// TwinCAT 3 PLC project PLC
// ProgramVersion: 3.1.4024.0
// libraries:
//   EfficientIO Communicator, * (EfficientIO)
//   EfficientIO Energy Basic, * (EfficientIO)
//   EfficientIO ModbusTCP, * (EfficientIO)
//   Lynus Energy ModbusRTU, * (Lynus AG)
//   Lynus Persistent Data V1, * (Lynus AG)
//   Lynus Standards, * (EfficientIO)
//   Tc2_Math, * (Beckhoff Automation GmbH)
//   Tc2_MBus, * (Beckhoff Automation GmbH)
//   Tc2_Standard, * (Beckhoff Automation GmbH)
//   Tc2_System, * (Beckhoff Automation GmbH)
//   Tc2_Utilities, * (Beckhoff Automation GmbH)
//   Tc3_JsonXml, * (Beckhoff Automation GmbH)
//   Tc3_Module, * (Beckhoff Automation GmbH)
// project tree:
//   / Fast_Task.TcTTO, Middle_Task.TcTTO, Slow_Task.TcTTO (not stored)
//   FB/ FB_CoE_EL3443.TcPOU (not stored), FB_EM_Beckhoff_EL3443.TcPOU (not stored), FB_TimeSwitch_V2.TcPOU
//   POUs/ prgComEffIO.TcPOU, prgEM.TcPOU, prgEMS.TcPOU, prgGrid.TcPOU, prgHouse.TcPOU, prgPersistent.TcPOU (not stored), prgRWEffIO.TcPOU (not stored), prgSystemTime.TcPOU (not stored), prgVarEffIO.TcPOU (not stored)
// real-time tasks:
//   TASK Fast_Task: cycle T#8ms, priority 8, ADS port 350
//   TASK Middle_Task: cycle T#10ms, priority 10, ADS port 351
//   TASK Slow_Task: cycle T#20ms, priority 20, ADS port 352
// I/O:
//   DEVICE Gerät 1 (Beckhoff CCAT)
//   DEVICE Gerät 2 (EtherCAT), AmsNetId 5.100.32.125.3.1
//     Klemme 1 (EK1200) [EK1200-5000 EtherCAT Netzteil (2A E-Bus)]
//       Klemme 2 (EL3443) [EL3443 3K. Leistungsmessung]
//       Klemme 3 (EL2652) [EL2652 2K. Relais Ausgang, Wechsler (230V AC / 30V DC)]
//       Klemme 4 (EL2652) [EL2652 2K. Relais Ausgang, Wechsler (230V AC / 30V DC)]
//       Klemme 5 (EL2652) [EL2652 2K. Relais Ausgang, Wechsler (230V AC / 30V DC)]
//       Klemme 6 (EL2652) [EL2652 2K. Relais Ausgang, Wechsler (230V AC / 30V DC)]
//       Klemme 7 (EL9011) [EL9011 Endklemme]
// variable links:
//   PLC/PLC Instance <-> Device 2 (EtherCAT)/Term 1 (EK1200)/Term 2 (EL3443)
//     Middle_Task Inputs/prgGrid.lrActivePowerTotal <-> Total Active/Active Power
//     Middle_Task Inputs/prgGrid.lrGrid_Current_L1 <-> L1 Basic/Current
//     Middle_Task Inputs/prgGrid.lrGrid_Current_L2 <-> L2 Basic/Current
//     Middle_Task Inputs/prgGrid.lrGrid_Current_L3 <-> L3 Basic/Current
//     Middle_Task Inputs/prgGrid.lrGrid_Power_L1 <-> L1 Power/Active Power
//     Middle_Task Inputs/prgGrid.lrGrid_Power_L2 <-> L2 Power/Active Power
//     Middle_Task Inputs/prgGrid.lrGrid_Power_L3 <-> L3 Power/Active Power
//     Middle_Task Inputs/prgGrid.lrGrid_Voltage_L1 <-> L1 Basic/Voltage
//     Middle_Task Inputs/prgGrid.lrGrid_Voltage_L2 <-> L2 Basic/Voltage
//     Middle_Task Inputs/prgGrid.lrGrid_Voltage_L3 <-> L3 Basic/Voltage
//   PLC/PLC Instance <-> Device 2 (EtherCAT)/Term 1 (EK1200)/Term 3 (EL2652)
//     Middle_Task Outputs/prgEM.Boiler <-> Channel 2/Output
//     Middle_Task Outputs/prgEM.KaffeMaschine <-> Channel 1/Output
//   PLC/PLC Instance <-> Device 2 (EtherCAT)/Term 1 (EK1200)/Term 4 (EL2652)
//     Middle_Task Outputs/prgEM.Heizregister <-> Channel 2/Output
//     Middle_Task Outputs/prgEM.Reklame <-> Channel 1/Output
//   PLC/PLC Instance <-> Device 2 (EtherCAT)/Term 1 (EK1200)/Term 5 (EL2652)
//     Middle_Task Outputs/prgEM.Abluft <-> Channel 2/Output
//     Middle_Task Outputs/prgEM.Zuluft <-> Channel 1/Output

CONFIGURATION PLC
    RESOURCE PLC ON TwinCAT3
        TASK Fast_Task(INTERVAL := T#8ms, PRIORITY := 8);
        TASK Middle_Task(INTERVAL := T#10ms, PRIORITY := 10);
        PROGRAM prgVarEffIO WITH Fast_Task : prgVarEffIO;
        PROGRAM prgRWEffIO WITH Fast_Task : prgRWEffIO;
        PROGRAM prgPersistent WITH Middle_Task : prgPersistent;
        PROGRAM prgGrid WITH Middle_Task : prgGrid;
        PROGRAM prgEM WITH Middle_Task : prgEM;
    END_RESOURCE
END_CONFIGURATION

// ---- POUs/prgGrid.TcPOU
PROGRAM prgGrid
VAR
	fbKBusState					: FB_K_Bus_State;
	fbGrid						: FB_EM_Beckhoff_KL3403;
	uint_KBusState				: UINT;							//{#lynus.ag#()}
	fbGridCounter				: FB_EnergyCounter;
	lrGridPower					: LREAL;								//{#lynus.ag#()}
	lrVoltage_L1N				: LREAL;								//{#lynus.ag#()}
	lrVoltage_L2N				: LREAL;								//{#lynus.ag#()}
	lrVoltage_L3N				: LREAL;								//{#lynus.ag#()}
	
	lrGrid_Voltage_L1  	AT %I* 	: REAL;									//{#lynus.ag#()}
    lrGrid_Current_L1 	AT %I* 	: REAL;									//{#lynus.ag#()}
	lrGrid_Power_L1		AT %I* 	: REAL;									//{#lynus.ag#()}
	lrGrid_Voltage_L2  	AT %I* 	: REAL;									//{#lynus.ag#()}
    lrGrid_Current_L2 	AT %I* 	: REAL;									//{#lynus.ag#()}
	lrGrid_Power_L2		AT %I* 	: REAL;									//{#lynus.ag#()}
	lrGrid_Voltage_L3  	AT %I* 	: REAL;									//{#lynus.ag#()}
    lrGrid_Current_L3 	AT %I* 	: REAL;									//{#lynus.ag#()}
	lrGrid_Power_L3		AT %I* 	: REAL;									//{#lynus.ag#()}
	lrActivePowerTotal	AT %I*	: REAL;									//{#lynus.ag#()}
	

	Test : REAL;

	Grid_Voltage_L1  	: REAL;						

END_VAR
VAR PERSISTENT
	rSizeGridConn				: REAL;									//{#lynus.ag#()}
	lrCounterGridProd			: LREAL;								//{#lynus.ag#()}
	lrCounterGridCons			: LREAL;								//{#lynus.ag#()}
END_VAR

//The mapping of this function must be linked with the K-Bus State in the E/A Part
fbKBusState(	uiKBusState_OUT=> , 
				b_Kbus_notOk=> , 
				word_ErrorCount=> );
				
//Variablen werden verwendet -> Middle Task
Test:= lrGrid_Voltage_L1;
Test:= lrGrid_Current_L1;
Test:= lrGrid_Power_L1;
Test:= lrGrid_Voltage_L2;
Test:= lrGrid_Current_L2;
Test:= lrGrid_Power_L2;
Test:= lrGrid_Voltage_L3;
Test:= lrGrid_Current_L3;
Test:= lrGrid_Power_L3;
Test:= lrActivePowerTotal;

//The mapping of this function must be linked with the KL3443 in the E/A Part
//UV1
fbGrid(
	bEnable:= FALSE, 
	bChannel1Invers:= FALSE,				//Invert power data when transformer are mounted upside down
	bChannel2Invers:= FALSE,				// CT seems to be wired the wrong wy around
	bChannel3Invers:= FALSE,
	uiCurrentTransformerRatioL1:= 300, 		//Transformer ratio on the secondary side
	uiCurrentTransformerRatioL2:= 300, 
	uiCurrentTransformerRatioL3:= 300, 
	uiKBusState_IN:= fbKBusState.uiKBusState_OUT, 
	stDataEMPower=> , 
	stDataEMCounter=> , 
	stDataEMPowerRealTime=> , 
	stDataEMCounterRealTime=> , 
	diNrOfEM_OUT=> );
	
uint_KBusState 	:=	fbKBusState.uiKBusState_OUT;
lrGridPower 	:= 	lrActivePowerTotal/1000;

// EnergyCounter
fbGridCounter(
	byActiveTariff:= 1, 
	lrPowerInput:= lrGridPower, 
	lrTotalCounterEnergy_Consumption=> , 
	lrTotalCounterEnergy_Production=> , 
	lrCounterEnergyT1_Consumption=> , 
	lrCounterEnergyT2_Consumption=> , 
	lrCounterEnergyT1_Production=> , 
	lrCounterEnergyT2_Production=> );

IF fbGridCounter.lrTotalCounterEnergy_Production > lrCounterGridProd THEN  	
		lrCounterGridProd := fbGridCounter.lrTotalCounterEnergy_Production;
END_IF

IF fbGridCounter.lrTotalCounterEnergy_Consumption > lrCounterGridCons THEN  	
	lrCounterGridCons := fbGridCounter.lrTotalCounterEnergy_Consumption;
END_IF

lrVoltage_L1N := fbGrid.stDataEMPower.lrVoltageL1N;
lrVoltage_L2N := fbGrid.stDataEMPower.lrVoltageL2N;
lrVoltage_L3N := fbGrid.stDataEMPower.lrVoltageL3N;

END_PROGRAM

// ---- POUs/prgEM.TcPOU
PROGRAM prgEM
VAR
	//Eingangsvariable: Aktueller Leistungswert aus prgGrid
    PowerValue 				: REAL := prgGrid.lrGridPower;
	Threshold 				: REAL := 35.0;  				//Schwelle zum Abschalten
	//Hysterese zum Vermeiden von schnellen Ein-/Ausschaltvorgängen
    Hysteresis 				: REAL := 5.0;
	//Zustandsvariablen zur Vermeidung von Schwingungen
    BoilerActive	 		: BOOL := TRUE;
    ReklameActive	 		: BOOL := TRUE;
	HeizregisterActive		: BOOL := TRUE;
    ZuluftActive	 		: BOOL := TRUE;
	AbluftActive	 		: BOOL := TRUE;
	//RELAI 1
	KaffeMaschine  	AT %Q* 	: BOOL;
	Boiler  		AT %Q* 	: BOOL;
	//RELAI 2
	Reklame  		AT %Q* 	: BOOL;
	Heizregister	AT %Q* 	: BOOL;
	//RELAI 3
	Zuluft  		AT %Q* 	: BOOL;
	Abluft	 		AT %Q* 	: BOOL;
	//RELAI 4 - OFFEN (Keine Anschlüsse)
	//RELAI4_CH1		AT %Q* 	: BOOL;
	//RELAI4_CH2		AT %Q* 	: BOOL;
	
	Test					:BOOL;
	
END_VAR

Test := KaffeMaschine;
Test := Boiler;
Test := Reklame;
Test := Heizregister;
Test := Zuluft;
Test := Abluft;
(* Logik zum Lastenmanagement mit einem Schwellenwert *)

(* Relais 1 CH 2 - Einschalten *)
IF PowerValue > Threshold AND BoilerActive THEN
    Boiler 			:= TRUE; 							//Relai wird eingeschalten um die Verbindung zu öffnen
    BoilerActive 	:= FALSE;
ELSIF PowerValue < (Threshold - Hysteresis) AND NOT BoilerActive THEN
    Boiler 			:= FALSE;  
    BoilerActive 	:= TRUE;
END_IF;
(*
(* Relais 2 CH1 - Einschalten *)
IF PowerValue > Threshold AND ReklameActive THEN
    Reklame 		:= TRUE; (* Relais 2 einschalten *)
    ReklameActive 	:= FALSE;
ELSIF PowerValue < (Threshold - Hysteresis) AND NOT ReklameActive THEN
    Reklame			:= FALSE;  (* Relais 2 ausschalten *)
    ReklameActive 	:= TRUE;
END_IF;
*)
(* Relais 2 CH2 - Einschalten *)
IF PowerValue > Threshold AND HeizregisterActive THEN
    Heizregister 		:= TRUE; (* Relais 2 einschalten *)
    HeizregisterActive 	:= FALSE;
ELSIF PowerValue < (Threshold - Hysteresis) AND NOT HeizregisterActive THEN
    Heizregister		:= FALSE;  (* Relais 2 ausschalten *)
    HeizregisterActive 	:= TRUE;
END_IF;

(* Relais 3 CH1 & CH2 - Einschalten *)
IF PowerValue > Threshold AND ZuluftActive AND AbluftActive THEN
    Zuluft := TRUE;
	Abluft := TRUE;
    ZuluftActive := FALSE;
	AbluftActive := FALSE;
ELSIF PowerValue < (Threshold - Hysteresis) AND NOT ZuluftActive AND NOT AbluftActive THEN
    Zuluft := FALSE;
	Abluft := FALSE;
	ZuluftActive := TRUE;
	AbluftActive := TRUE;
END_IF;

END_PROGRAM

// ---- FB/FB_TimeSwitch_V2.TcPOU
FUNCTION_BLOCK FB_TimeSwitch_V2
VAR_INPUT
	b_Enable: BOOL;
	b_StatusOn: BOOL;
	structSystemTime: timestruct;
	byte_MoFr_Open_Hour: BYTE;
	byte_MoFr_Open_Minute: BYTE;
	byte_MoFr_Close_Hour: BYTE;
	byte_MoFr_Close_Minute: BYTE;
	byte_Sa_Open_Hour: BYTE;
	byte_Sa_Open_Minute: BYTE;
	byte_Sa_Close_Hour: BYTE;
	byte_Sa_Close_Minute: BYTE;	
	byte_So_Open_Hour: BYTE;
	byte_So_Open_Minute: BYTE;
	byte_So_Close_Hour: BYTE;
	byte_So_Close_Minute: BYTE;
	real_Offset_Start: REAL;
	real_Offset_Stop: REAL;	
	b_On_Manual: BOOL;
	b_Off_Manual: BOOL;
END_VAR
VAR_OUTPUT
	b_Output_On: BOOL;
	b_Error: BOOL;
END_VAR
VAR
	TON_0: ton;
	byte_Day :BYTE;		// 0: Sunday, 1: Monday,....
	time_now             		: TIME;
	time_MoFr_Open             	: TIME;
	time_MoFr_Close             : TIME;
	time_Sa_Open             	: TIME;
	time_Sa_Close             	: TIME;
	time_So_Open             	: TIME;
	time_So_Close             	: TIME;
	

	RS_0: rs;
	R_TRIG_0: r_trig;
	R_TRIG_1: r_trig;
	dt_Test: DATE_AND_TIME;
	tod_test: TIME_OF_DAY;
	time_temp: TIME;
	time_Start_MoFr_Calc: TIME;
	time_Stop_MoFr_Calc: TIME;
	time_Start_Sa_Calc: TIME;
	time_Stop_Sa_Calc: TIME;
	time_Start_So_Calc: TIME;
	time_Stop_So_Calc: TIME;
	
	FB_WeeklyTimeSwitch_MoFr: FB_WeeklyTimeSwitch;
	FB_WeeklyTimeSwitch_Sa: FB_WeeklyTimeSwitch;
	FB_WeeklyTimeSwitch_So: FB_WeeklyTimeSwitch;
	RS_manu: rs;
	b_Auto_on: BOOL;

	R_TRIG_2: r_trig;
	R_TRIG_3: r_trig;
	F_TRIG_0: f_trig;
	R_TRIG_4: r_trig;
	R_TRIG_FirstCycle: r_trig;
	time_Zero             	: TIME;
	
END_VAR
VAR // added by the converter: edge detectors and wires of the graphical bodies
    _w1 : DATE_AND_TIME;
    _w2 : TIME_OF_DAY;
    _w3 : BOOL;
END_VAR

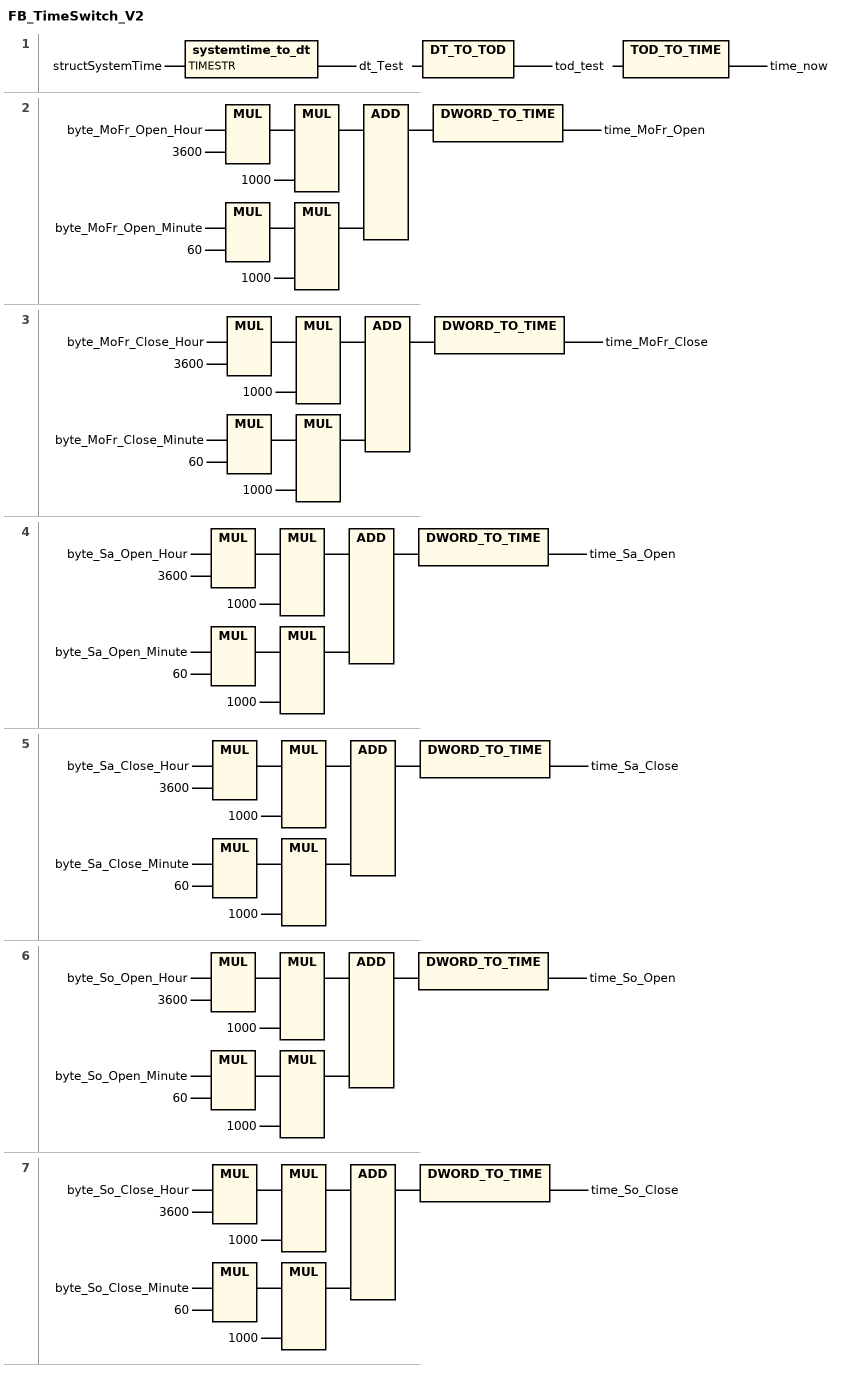
// NETWORK 1
_w1 := systemtime_to_dt(TIMESTR := structSystemTime);
dt_Test := _w1;
_w2 := DT_TO_TOD(_w1);
tod_test := _w2;
time_now := TOD_TO_TIME(_w2);

// NETWORK 2
time_MoFr_Open := DWORD_TO_TIME((byte_MoFr_Open_Hour * 3600) * 1000 + (byte_MoFr_Open_Minute * 60) * 1000);

// NETWORK 3
time_MoFr_Close := DWORD_TO_TIME((byte_MoFr_Close_Hour * 3600) * 1000 + (byte_MoFr_Close_Minute * 60) * 1000);

// NETWORK 4
time_Sa_Open := DWORD_TO_TIME((byte_Sa_Open_Hour * 3600) * 1000 + (byte_Sa_Open_Minute * 60) * 1000);

// NETWORK 5
time_Sa_Close := DWORD_TO_TIME((byte_Sa_Close_Hour * 3600) * 1000 + (byte_Sa_Close_Minute * 60) * 1000);

// NETWORK 6
time_So_Open := DWORD_TO_TIME((byte_So_Open_Hour * 3600) * 1000 + (byte_So_Open_Minute * 60) * 1000);

// NETWORK 7
time_So_Close := DWORD_TO_TIME((byte_So_Close_Hour * 3600) * 1000 + (byte_So_Close_Minute * 60) * 1000);

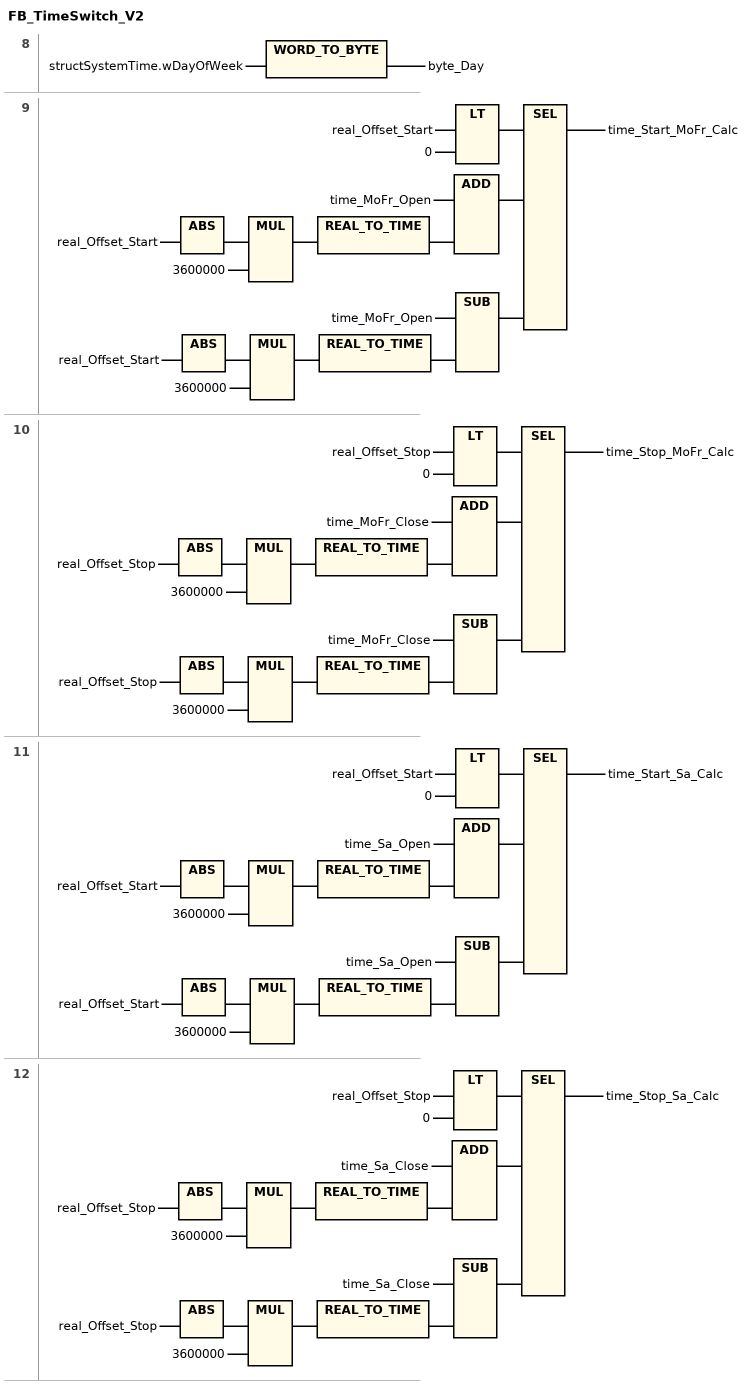
// NETWORK 8
byte_Day := WORD_TO_BYTE(structSystemTime.wDayOfWeek);

// NETWORK 9
time_Start_MoFr_Calc := SEL(real_Offset_Start < 0, time_MoFr_Open + REAL_TO_TIME(ABS(real_Offset_Start) * 3600000), time_MoFr_Open - REAL_TO_TIME(ABS(real_Offset_Start) * 3600000));

// NETWORK 10
time_Stop_MoFr_Calc := SEL(real_Offset_Stop < 0, time_MoFr_Close + REAL_TO_TIME(ABS(real_Offset_Stop) * 3600000), time_MoFr_Close - REAL_TO_TIME(ABS(real_Offset_Stop) * 3600000));

// NETWORK 11
time_Start_Sa_Calc := SEL(real_Offset_Start < 0, time_Sa_Open + REAL_TO_TIME(ABS(real_Offset_Start) * 3600000), time_Sa_Open - REAL_TO_TIME(ABS(real_Offset_Start) * 3600000));

// NETWORK 12
time_Stop_Sa_Calc := SEL(real_Offset_Stop < 0, time_Sa_Close + REAL_TO_TIME(ABS(real_Offset_Stop) * 3600000), time_Sa_Close - REAL_TO_TIME(ABS(real_Offset_Stop) * 3600000));

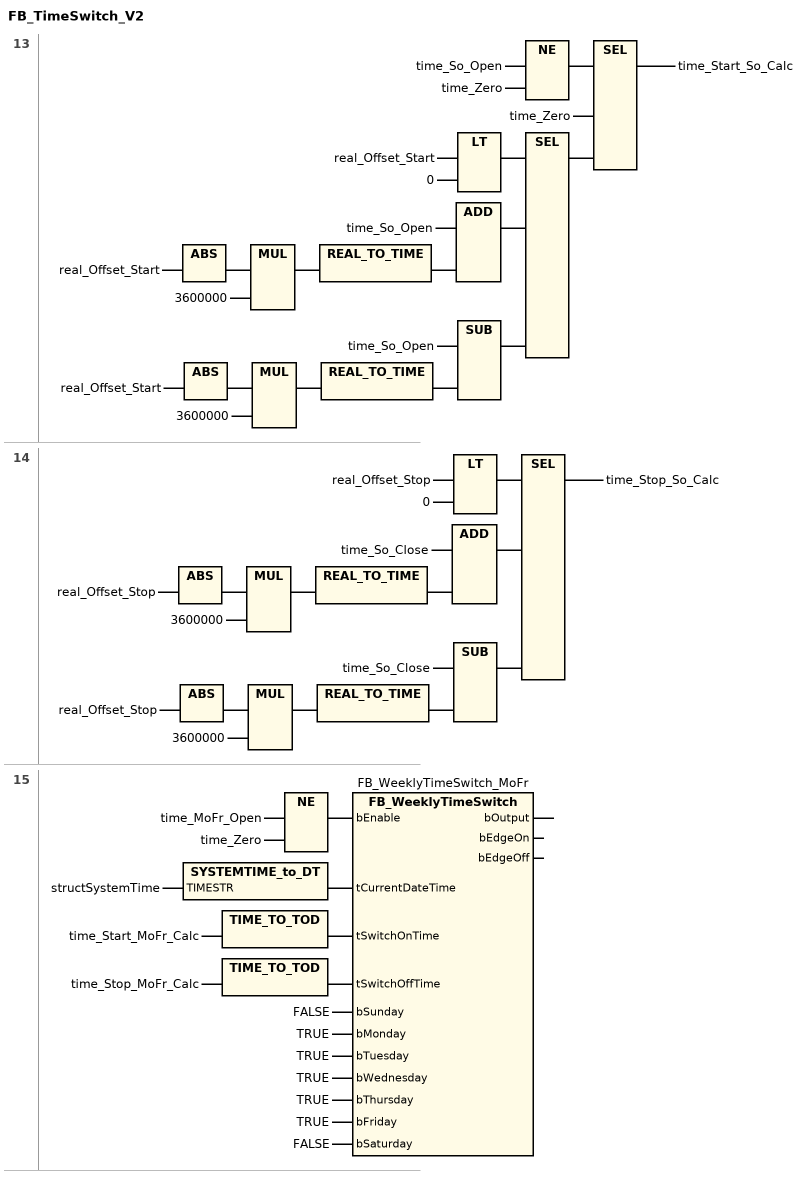
// NETWORK 13
time_Start_So_Calc := SEL(time_So_Open <> time_Zero, time_Zero, SEL(real_Offset_Start < 0, time_So_Open + REAL_TO_TIME(ABS(real_Offset_Start) * 3600000), time_So_Open - REAL_TO_TIME(ABS(real_Offset_Start) * 3600000)));

// NETWORK 14
time_Stop_So_Calc := SEL(real_Offset_Stop < 0, time_So_Close + REAL_TO_TIME(ABS(real_Offset_Stop) * 3600000), time_So_Close - REAL_TO_TIME(ABS(real_Offset_Stop) * 3600000));

// NETWORK 15
FB_WeeklyTimeSwitch_MoFr(
    bEnable := time_MoFr_Open <> time_Zero,
    tCurrentDateTime := SYSTEMTIME_to_DT(TIMESTR := structSystemTime),
    tSwitchOnTime := TIME_TO_TOD(time_Start_MoFr_Calc),
    tSwitchOffTime := TIME_TO_TOD(time_Stop_MoFr_Calc),
    bSunday := FALSE,
    bMonday := TRUE,
    bTuesday := TRUE,
    bWednesday := TRUE,
    bThursday := TRUE,
    bFriday := TRUE,
    bSaturday := FALSE); // FB_WeeklyTimeSwitch

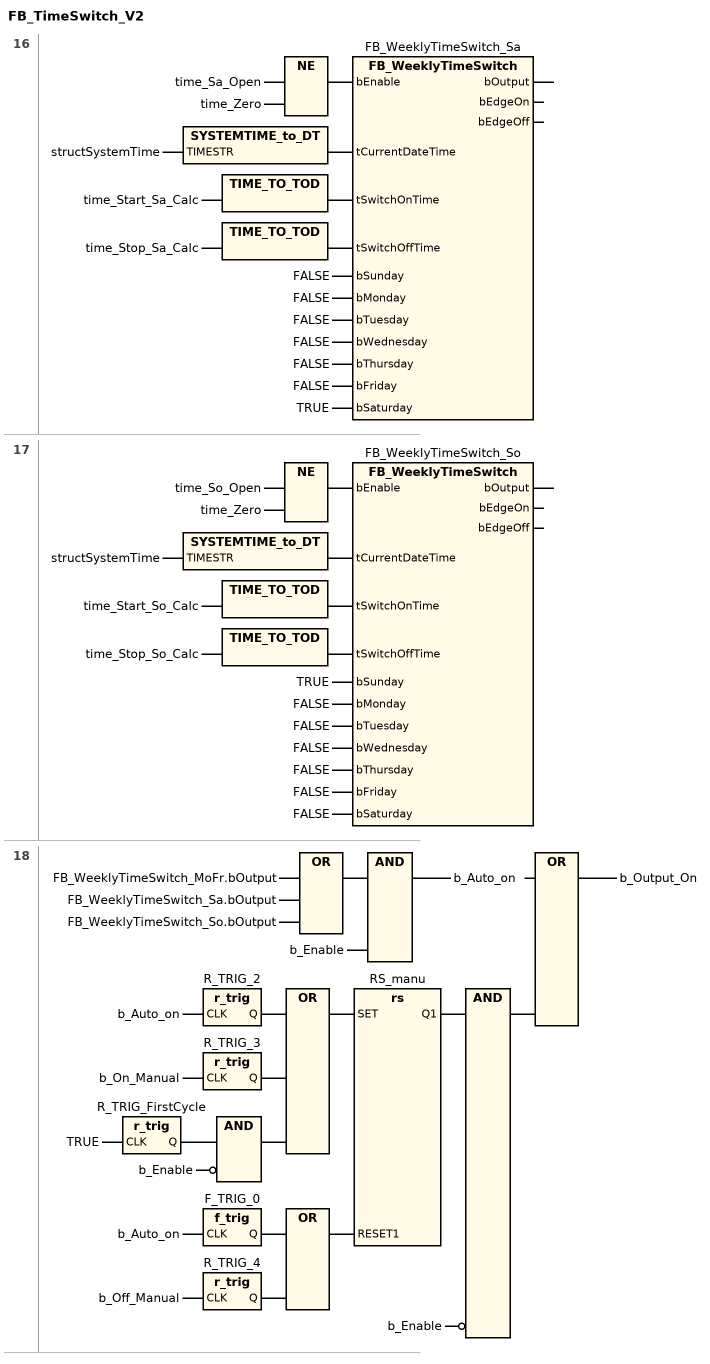
// NETWORK 16
FB_WeeklyTimeSwitch_Sa(
    bEnable := time_Sa_Open <> time_Zero,
    tCurrentDateTime := SYSTEMTIME_to_DT(TIMESTR := structSystemTime),
    tSwitchOnTime := TIME_TO_TOD(time_Start_Sa_Calc),
    tSwitchOffTime := TIME_TO_TOD(time_Stop_Sa_Calc),
    bSunday := FALSE,
    bMonday := FALSE,
    bTuesday := FALSE,
    bWednesday := FALSE,
    bThursday := FALSE,
    bFriday := FALSE,
    bSaturday := TRUE); // FB_WeeklyTimeSwitch

// NETWORK 17
FB_WeeklyTimeSwitch_So(
    bEnable := time_So_Open <> time_Zero,
    tCurrentDateTime := SYSTEMTIME_to_DT(TIMESTR := structSystemTime),
    tSwitchOnTime := TIME_TO_TOD(time_Start_So_Calc),
    tSwitchOffTime := TIME_TO_TOD(time_Stop_So_Calc),
    bSunday := TRUE,
    bMonday := FALSE,
    bTuesday := FALSE,
    bWednesday := FALSE,
    bThursday := FALSE,
    bFriday := FALSE,
    bSaturday := FALSE); // FB_WeeklyTimeSwitch

// NETWORK 18
_w3 := (FB_WeeklyTimeSwitch_MoFr.bOutput OR FB_WeeklyTimeSwitch_Sa.bOutput OR FB_WeeklyTimeSwitch_So.bOutput) AND b_Enable;
b_Auto_on := _w3;
R_TRIG_2(CLK := b_Auto_on); // r_trig
R_TRIG_3(CLK := b_On_Manual); // r_trig
R_TRIG_FirstCycle(CLK := TRUE); // r_trig
F_TRIG_0(CLK := b_Auto_on); // f_trig
R_TRIG_4(CLK := b_Off_Manual); // r_trig
RS_manu(SET := R_TRIG_2.Q OR R_TRIG_3.Q OR R_TRIG_FirstCycle.Q AND NOT b_Enable, RESET1 := F_TRIG_0.Q OR R_TRIG_4.Q); // rs
b_Output_On := _w3 OR RS_manu.Q1 AND NOT b_Enable;

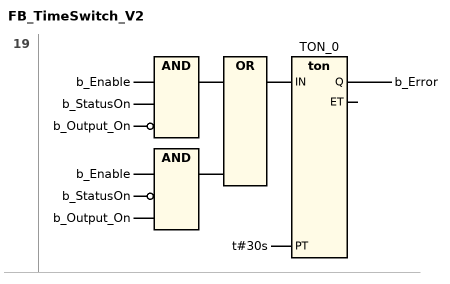
// NETWORK 19
TON_0(IN := b_Enable AND b_StatusOn AND NOT b_Output_On OR b_Enable AND NOT b_StatusOn AND b_Output_On, PT := t#30s); // ton
b_Error := TON_0.Q;

END_FUNCTION_BLOCK

// ---- POUs/prgComEffIO.TcPOU
PROGRAM prgComEffIO
VAR
	fbCom		: FB_MqttCommunicator_V5;
END_VAR

// CX-7BDACD
fbCom(
	bConnect:= TRUE, 
	strAuthKey := 'ENE87365342998',
	sUserName:= 'a4398363-713f-45e4-8f12-13b95d7f2606', 
	sUserPassword:= '196c948c-aabd-4764-8be4-f15873a2b8fa', 
	eSavePositionCertificate:= eSavePositionOnPLC.ePostionHardDisk,
	time_HeartBeat_sec:= T#50S, 
	bConnected=> , 
	bError=> , 
	hrErrorCode=> , 
	eConnectionState=> , 
	eErrorMessage_Out=> );

END_PROGRAM

// ---- POUs/prgEMS.TcPOU
PROGRAM prgEMS
VAR
	FB_TimeSwitch_CH1: FB_TimeSwitch_v2;
	FB_TimeSwitch_CH2: FB_TimeSwitch_v2;
	FB_TimeSwitch_CH3: FB_TimeSwitch_v2;
	FB_TimeSwitch_CH4: FB_TimeSwitch_v2;
	FB_TimeSwitch_CH5: FB_TimeSwitch_v2;	// outside light
	FB_TimeSwitch_CH6: FB_TimeSwitch_v2;	// Coffee maschine
	FB_TimeSwitch_CH7: FB_TimeSwitch_v2;	// Ventilation
	FB_TimeSwitch_CH8: FB_TimeSwitch_v2;	// Coffee maschine2
	
	b_Manual_On_CH1		: BOOL;						//{#lynus.ag#()}
	b_Manual_Off_CH1	: BOOL;						//{#lynus.ag#()}
	b_Manual_On_CH2		: BOOL;						//{#lynus.ag#()}
	b_Manual_Off_CH2	: BOOL;						//{#lynus.ag#()}
	b_Manual_On_CH3		: BOOL;						//{#lynus.ag#()}
	b_Manual_Off_CH3	: BOOL;						//{#lynus.ag#()}
	b_Manual_On_CH4		: BOOL;						//{#lynus.ag#()}
	b_Manual_Off_CH4	: BOOL;						//{#lynus.ag#()}
	b_Manual_On_CH5		: BOOL;						//{#lynus.ag#()}
	b_Manual_Off_CH5	: BOOL;						//{#lynus.ag#()}
	b_Manual_On_Coffee_CH6		: BOOL;						//{#lynus.ag#()}
	b_Manual_Off_Coffee_CH6		: BOOL;						//{#lynus.ag#()}
	b_Manual_On_Vent_CH7		: BOOL;						//{#lynus.ag#()}
	b_Manual_Off_Vent_CH7		: BOOL;						//{#lynus.ag#()}
	b_Manual_On_Coffee2_CH8		: BOOL;						//{#lynus.ag#()}
	b_Manual_Off_Coffee2_CH8	: BOOL;						//{#lynus.ag#()}

	fbCalcSunriseSunset   		: FB_CalcSunriseSunset;
	todSunrise            		: TOD;
	todSunset             		: TOD;
	fb_GetTimeZoneInfo	:FB_GetTimeZoneInformation;
	b_firstCycle: BOOL;
	RS_Outsidelight: RS;
	r_trig_on: R_trig;
	r_trig_off: R_trig;
	b_Out_CH1: BOOL;
	b_Out_CH2: BOOL;
	b_Out_CH3: BOOL;
	b_Out_CH4: BOOL;
	b_Out_CH5: BOOL;
	b_Out_CH6: BOOL;
	b_Out_CH7: BOOL;		
	b_Out_CH8: BOOL;		
	b_LoadOn_CH1	: BOOL;						//{#lynus.ag#()}
	b_LoadOn_CH2	: BOOL;						//{#lynus.ag#()}
	b_LoadOn_CH3	: BOOL;						//{#lynus.ag#()}
	b_LoadOn_CH4	: BOOL;						//{#lynus.ag#()}
	b_LoadOn_CH5	: BOOL;						//{#lynus.ag#()}
	b_LoadOn_CH6	: BOOL;						//{#lynus.ag#()}
	b_LoadOn_CH7	: BOOL;						//{#lynus.ag#()}
	b_LoadOn_CH8	: BOOL;						//{#lynus.ag#()}
END_VAR
VAR_INPUT
	fDegreeOfLongitude 	:LREAL;
	fDegreeOfLatitude	:LREAL;
	b_Input_KeySwitch		: BOOL;						//{#lynus.ag#()}
	b_Input_Spare			: BOOL;						//{#lynus.ag#()}
	m_UnderGroundMode		: BOOL;						//{#lynus.ag#()}
	int_test:INT;
END_VAR
VAR PERSISTENT
// opening hours
	byte_MoFr_Open_Hour		:BYTE;					//{#lynus.ag#()}
	byte_MoFr_Open_Minute	:BYTE;					//{#lynus.ag#()}
	byte_MoFr_Close_Hour	:BYTE;					//{#lynus.ag#()}
	byte_MoFr_Close_Minute	:BYTE;					//{#lynus.ag#()}
	byte_Sa_Open_Hour		:BYTE;					//{#lynus.ag#()}
	byte_Sa_Open_Minute		:BYTE;					//{#lynus.ag#()}
	byte_Sa_Close_Hour		:BYTE;					//{#lynus.ag#()}
	byte_Sa_Close_Minute	:BYTE;					//{#lynus.ag#()}
	byte_So_Open_Hour		:BYTE;					//{#lynus.ag#()}
	byte_So_Open_Minute		:BYTE;					//{#lynus.ag#()}
	byte_So_Close_Hour		:BYTE;					//{#lynus.ag#()}
	byte_So_Close_Minute	:BYTE;					//{#lynus.ag#()}
// offset CH1 in hours			
	b_Enable_Control_CH1		:BOOL;				//{#lynus.ag#()}
	real_Offset_Start_CH1		:REAL;				//{#lynus.ag#()}
	real_Offset_Stop_CH1		:REAL;				//{#lynus.ag#()}
// offset CH2 in hours			
	b_Enable_Control_CH2		:BOOL;				//{#lynus.ag#()}
	real_Offset_Start_CH2		:REAL;				//{#lynus.ag#()}
	real_Offset_Stop_CH2		:REAL;				//{#lynus.ag#()}
// offset CH3 in hours			
	b_Enable_Control_CH3		:BOOL;				//{#lynus.ag#()}
	real_Offset_Start_CH3		:REAL;				//{#lynus.ag#()}
	real_Offset_Stop_CH3		:REAL;				//{#lynus.ag#()}
// offset CH4 in hours			
	b_Enable_Control_CH4		:BOOL;				//{#lynus.ag#()}
	real_Offset_Start_CH4		:REAL;				//{#lynus.ag#()}
	real_Offset_Stop_CH4		:REAL;				//{#lynus.ag#()}
// offset CH5 in hours			
	b_Enable_Control_CH5		:BOOL;				//{#lynus.ag#()}
	real_Offset_Start_CH5		:REAL;				//{#lynus.ag#()}
	real_Offset_Stop_CH5		:REAL;				//{#lynus.ag#()}
// offset CH6 in hours			
	b_Enable_Control_Coffee_CH6	:BOOL;				//{#lynus.ag#()}
	real_Offset_Start_Coffee_CH6:REAL;				//{#lynus.ag#()}
	real_Offset_Stop_Coffee_CH6	:REAL;				//{#lynus.ag#()}
// offset CH7 in hours			
	b_Enable_Control_Vent_CH7	:BOOL;				//{#lynus.ag#()}
	real_Offset_Start_CH7		:REAL;				//{#lynus.ag#()}
	real_Offset_Stop_CH7		:REAL;				//{#lynus.ag#()}
// offset CH8 in hours			
	b_Enable_Control_Coffee2_CH8	:BOOL;				//{#lynus.ag#()}
	real_Offset_Start_Coffee2_CH8	:REAL;				//{#lynus.ag#()}
	real_Offset_Stop_Coffee2_CH8	:REAL;				//{#lynus.ag#()}
END_VAR


FB_TimeSwitch_CH1(
	b_Enable:= b_Enable_Control_CH1, 
	b_StatusOn:= NOT b_Out_CH1, 
	structSystemTime:=prgSystemTime.structSystemTime , 
	byte_MoFr_Open_Hour:= byte_MoFr_Open_Hour , 
	byte_MoFr_Open_Minute:= byte_MoFr_Open_Minute, 
	byte_MoFr_Close_Hour:= byte_MoFr_Close_Hour , 
	byte_MoFr_Close_Minute:= byte_MoFr_Close_Minute, 
	byte_Sa_Open_Hour:= byte_Sa_Open_Hour, 
	byte_Sa_Open_Minute:= byte_Sa_Open_Minute , 
	byte_Sa_Close_Hour:= byte_Sa_Close_Hour , 
	byte_Sa_Close_Minute:= byte_Sa_Close_Minute, 
	byte_So_Open_Hour:= byte_So_Open_Hour, 
	byte_So_Open_Minute:= byte_So_Open_Minute, 
	byte_So_Close_Hour:= byte_So_Close_Hour, 
	byte_So_Close_Minute:= byte_So_Close_Minute, 
	real_Offset_Start:= real_Offset_Start_CH1 , 
	real_Offset_Stop:= real_Offset_Stop_CH1 , 
	b_On_Manual:= b_Manual_On_CH1, 
	b_Off_Manual:= b_Manual_Off_CH1, 
	b_Output_On=> b_LoadOn_CH1, 
	b_Error=> );
b_Out_CH1 := NOT FB_TimeSwitch_CH1.b_Output_On;

FB_TimeSwitch_CH2(
	b_Enable:= b_Enable_Control_CH2, 
	b_StatusOn:= NOT b_Out_CH2, 
	structSystemTime:=prgSystemTime.structSystemTime , 
	byte_MoFr_Open_Hour:= byte_MoFr_Open_Hour , 
	byte_MoFr_Open_Minute:= byte_MoFr_Open_Minute, 
	byte_MoFr_Close_Hour:= byte_MoFr_Close_Hour , 
	byte_MoFr_Close_Minute:= byte_MoFr_Close_Minute, 
	byte_Sa_Open_Hour:= byte_Sa_Open_Hour, 
	byte_Sa_Open_Minute:= byte_Sa_Open_Minute , 
	byte_Sa_Close_Hour:= byte_Sa_Close_Hour , 
	byte_Sa_Close_Minute:= byte_Sa_Close_Minute, 
	byte_So_Open_Hour:= byte_So_Open_Hour, 
	byte_So_Open_Minute:= byte_So_Open_Minute, 
	byte_So_Close_Hour:= byte_So_Close_Hour, 
	byte_So_Close_Minute:= byte_So_Close_Minute, 
	real_Offset_Start:= real_Offset_Start_CH2 , 
	real_Offset_Stop:= real_Offset_Stop_CH2 , 
	b_On_Manual:= b_Manual_On_CH2, 
	b_Off_Manual:= b_Manual_Off_CH2, 
	b_Output_On=> b_LoadOn_CH2, 
	b_Error=> );
b_Out_CH2 := NOT FB_TimeSwitch_CH2.b_Output_On;

FB_TimeSwitch_CH3(
	b_Enable:= b_Enable_Control_CH3, 
	b_StatusOn:= NOT b_Out_CH3, 
	structSystemTime:=prgSystemTime.structSystemTime , 
	byte_MoFr_Open_Hour:= byte_MoFr_Open_Hour , 
	byte_MoFr_Open_Minute:= byte_MoFr_Open_Minute, 
	byte_MoFr_Close_Hour:= byte_MoFr_Close_Hour , 
	byte_MoFr_Close_Minute:= byte_MoFr_Close_Minute, 
	byte_Sa_Open_Hour:= byte_Sa_Open_Hour, 
	byte_Sa_Open_Minute:= byte_Sa_Open_Minute , 
	byte_Sa_Close_Hour:= byte_Sa_Close_Hour , 
	byte_Sa_Close_Minute:= byte_Sa_Close_Minute, 
	byte_So_Open_Hour:= byte_So_Open_Hour, 
	byte_So_Open_Minute:= byte_So_Open_Minute, 
	byte_So_Close_Hour:= byte_So_Close_Hour, 
	byte_So_Close_Minute:= byte_So_Close_Minute, 
	real_Offset_Start:= real_Offset_Start_CH3 , 
	real_Offset_Stop:= real_Offset_Stop_CH3 , 
	b_On_Manual:= b_Manual_On_CH3, 
	b_Off_Manual:= b_Manual_Off_CH3, 
	b_Output_On=> b_LoadOn_CH3, 
	b_Error=> );
b_Out_CH3 := NOT FB_TimeSwitch_CH3.b_Output_On;
	
FB_TimeSwitch_CH4(
	b_Enable:= b_Enable_Control_CH4, 
	b_StatusOn:= NOT b_Out_CH4, 
	structSystemTime:=prgSystemTime.structSystemTime , 
	byte_MoFr_Open_Hour:= byte_MoFr_Open_Hour , 
	byte_MoFr_Open_Minute:= byte_MoFr_Open_Minute, 
	byte_MoFr_Close_Hour:= byte_MoFr_Close_Hour , 
	byte_MoFr_Close_Minute:= byte_MoFr_Close_Minute, 
	byte_Sa_Open_Hour:= byte_Sa_Open_Hour, 
	byte_Sa_Open_Minute:= byte_Sa_Open_Minute , 
	byte_Sa_Close_Hour:= byte_Sa_Close_Hour , 
	byte_Sa_Close_Minute:= byte_Sa_Close_Minute, 
	byte_So_Open_Hour:= byte_So_Open_Hour, 
	byte_So_Open_Minute:= byte_So_Open_Minute, 
	byte_So_Close_Hour:= byte_So_Close_Hour, 
	byte_So_Close_Minute:= byte_So_Close_Minute, 
	real_Offset_Start:= real_Offset_Start_CH4 , 
	real_Offset_Stop:= real_Offset_Stop_CH4 , 
	b_On_Manual:= b_Manual_On_CH4, 
	b_Off_Manual:= b_Manual_Off_CH4, 
	b_Output_On=> b_LoadOn_CH4 ,
	b_Error=> );
b_Out_CH4 := NOT FB_TimeSwitch_CH4.b_Output_On;
	
FB_TimeSwitch_CH5(
	b_Enable:= b_Enable_Control_CH5, 
	b_StatusOn:= NOT b_Out_CH5, 
	structSystemTime:=prgSystemTime.structSystemTime , 
	byte_MoFr_Open_Hour:= byte_MoFr_Open_Hour , 
	byte_MoFr_Open_Minute:= byte_MoFr_Open_Minute, 
	byte_MoFr_Close_Hour:= byte_MoFr_Close_Hour , 
	byte_MoFr_Close_Minute:= byte_MoFr_Close_Minute, 
	byte_Sa_Open_Hour:= byte_Sa_Open_Hour, 
	byte_Sa_Open_Minute:= byte_Sa_Open_Minute , 
	byte_Sa_Close_Hour:= byte_Sa_Close_Hour , 
	byte_Sa_Close_Minute:= byte_Sa_Close_Minute, 
	byte_So_Open_Hour:= byte_So_Open_Hour, 
	byte_So_Open_Minute:= byte_So_Open_Minute, 
	byte_So_Close_Hour:= byte_So_Close_Hour, 
	byte_So_Close_Minute:= byte_So_Close_Minute, 
	real_Offset_Start:= real_Offset_Start_CH5 , 
	real_Offset_Stop:= real_Offset_Stop_CH5 , 
	b_On_Manual:= b_Manual_On_CH5, 
	b_Off_Manual:= b_Manual_Off_CH5, 
	b_Output_On=>  , 
	b_Error=> );
//b_Out_CH5 := NOT FB_TimeSwitch_CH5.b_Output_On; 		Outside light, done below
	
FB_TimeSwitch_CH6(
	b_Enable:= b_Enable_Control_Coffee_CH6, 
	b_StatusOn:= NOT b_Out_CH6, 
	structSystemTime:=prgSystemTime.structSystemTime , 
	byte_MoFr_Open_Hour:= byte_MoFr_Open_Hour , 
	byte_MoFr_Open_Minute:= byte_MoFr_Open_Minute, 
	byte_MoFr_Close_Hour:= byte_MoFr_Close_Hour , 
	byte_MoFr_Close_Minute:= byte_MoFr_Close_Minute, 
	byte_Sa_Open_Hour:= byte_Sa_Open_Hour, 
	byte_Sa_Open_Minute:= byte_Sa_Open_Minute , 
	byte_Sa_Close_Hour:= byte_Sa_Close_Hour , 
	byte_Sa_Close_Minute:= byte_Sa_Close_Minute, 
	byte_So_Open_Hour:= byte_So_Open_Hour, 
	byte_So_Open_Minute:= byte_So_Open_Minute, 
	byte_So_Close_Hour:= byte_So_Close_Hour, 
	byte_So_Close_Minute:= byte_So_Close_Minute, 
	real_Offset_Start:= real_Offset_Start_Coffee_CH6 , 
	real_Offset_Stop:= real_Offset_Stop_Coffee_CH6 , 
	b_On_Manual:= b_Manual_On_Coffee_CH6, 
	b_Off_Manual:= b_Manual_Off_Coffee_CH6, 
	b_Output_On=> b_LoadOn_CH6, 
	b_Error=> );
b_Out_CH6 := NOT FB_TimeSwitch_CH6.b_Output_On;
	
FB_TimeSwitch_CH7(
	b_Enable:= b_Enable_Control_Vent_CH7, 
	b_StatusOn:= NOT b_Out_CH7, 
	structSystemTime:=prgSystemTime.structSystemTime , 
	byte_MoFr_Open_Hour:= byte_MoFr_Open_Hour , 
	byte_MoFr_Open_Minute:= byte_MoFr_Open_Minute, 
	byte_MoFr_Close_Hour:= byte_MoFr_Close_Hour , 
	byte_MoFr_Close_Minute:= byte_MoFr_Close_Minute, 
	byte_Sa_Open_Hour:= byte_Sa_Open_Hour, 
	byte_Sa_Open_Minute:= byte_Sa_Open_Minute , 
	byte_Sa_Close_Hour:= byte_Sa_Close_Hour , 
	byte_Sa_Close_Minute:= byte_Sa_Close_Minute, 
	byte_So_Open_Hour:= byte_So_Open_Hour, 
	byte_So_Open_Minute:= byte_So_Open_Minute, 
	byte_So_Close_Hour:= byte_So_Close_Hour, 
	byte_So_Close_Minute:= byte_So_Close_Minute, 
	real_Offset_Start:= real_Offset_Start_CH7 , 
	real_Offset_Stop:= real_Offset_Stop_CH7 , 
	b_On_Manual:= b_Manual_On_Vent_CH7, 
	b_Off_Manual:= b_Manual_Off_Vent_CH7, 
	b_Output_On=> b_LoadOn_CH7, 
	b_Error=> );
b_Out_CH7 := NOT FB_TimeSwitch_CH7.b_Output_On;
	
	
// calculate sunset / sunrise
// find out the time details	
IF fDegreeOfLongitude= 0 OR fDegreeOfLatitude= 0 THEN 
	fDegreeOfLongitude := 16.3731;   (* Longitude of Vienna *)
	fDegreeOfLatitude := 48.2083;   (* Latitude of Vienna*)
END_IF
fb_GetTimeZoneInfo(
	sNetID:= '', 
	bExecute:= prgSystemTime.structSystemTime.wHour = 4 OR NOT b_firstCycle, 
	tTimeout:= T#5S, 
	bBusy=> , 
	bError=> , 
	nErrID=> , 
	tzID=> , 
	tzInfo=> );
b_firstCycle := TRUE;


fbCalcSunriseSunset(
	fDegreeOfLongitude :=,
	fDegreeOfLatitude := ,
	fReferenceMeridian := SEL( fb_GetTimeZoneInfo.tzID = eTimeZoneID_Daylight ,15,30),  (* Central European Time 15 Winter Timer / 30 Summer Time *)
	dCurrentDate := DT_TO_DATE(SYSTEMTIME_TO_Dt (prgSystemTime.structSystemTime)),
	todSunrise => todSunrise,
	todSunset => todSunset);
	
r_trig_on (clk := (FB_TimeSwitch_CH5.b_Output_On AND (DT_TO_TOD(systemtime_to_dt(prgSystemTime.structSystemTime))< (todSunrise +  T#1H))) OR (FB_TimeSwitch_CH5.b_Output_On AND m_UnderGroundMode));
r_trig_off (clk := NOT FB_TimeSwitch_CH5.b_Output_On);

RS_Outsidelight(	Set := r_trig_on.Q OR ((todSunset - T#2H) =  DT_TO_TOD(systemtime_to_dt(prgSystemTime.structSystemTime)) AND FB_TimeSwitch_CH5.b_Output_On AND NOT m_UnderGroundMode) OR b_Manual_On_CH5 ,
					Reset1 := r_trig_off.Q OR (((todSunrise +  T#1H)= DT_TO_TOD(systemtime_to_dt(prgSystemTime.structSystemTime))) AND NOT m_UnderGroundMode) OR b_Manual_Off_CH5,
					Q1 => b_LoadOn_CH5 );		
b_Out_CH5	:= NOT b_LoadOn_CH5;
	
FB_TimeSwitch_CH8(
	b_Enable:= b_Enable_Control_Coffee2_CH8, 
	b_StatusOn:= NOT b_Out_CH8, 
	structSystemTime:=prgSystemTime.structSystemTime , 
	byte_MoFr_Open_Hour:= byte_MoFr_Open_Hour , 
	byte_MoFr_Open_Minute:= byte_MoFr_Open_Minute, 
	byte_MoFr_Close_Hour:= byte_MoFr_Close_Hour , 
	byte_MoFr_Close_Minute:= byte_MoFr_Close_Minute, 
	byte_Sa_Open_Hour:= byte_Sa_Open_Hour, 
	byte_Sa_Open_Minute:= byte_Sa_Open_Minute , 
	byte_Sa_Close_Hour:= byte_Sa_Close_Hour , 
	byte_Sa_Close_Minute:= byte_Sa_Close_Minute, 
	byte_So_Open_Hour:= byte_So_Open_Hour, 
	byte_So_Open_Minute:= byte_So_Open_Minute, 
	byte_So_Close_Hour:= byte_So_Close_Hour, 
	byte_So_Close_Minute:= byte_So_Close_Minute, 
	real_Offset_Start:= real_Offset_Start_Coffee2_CH8 , 
	real_Offset_Stop:= real_Offset_Stop_Coffee2_CH8 , 
	b_On_Manual:= b_Manual_On_Coffee2_CH8, 
	b_Off_Manual:= b_Manual_Off_Coffee2_CH8, 
	b_Output_On=> b_LoadOn_CH8, 
	b_Error=> );
b_Out_CH8 := NOT FB_TimeSwitch_CH8.b_Output_On;

END_PROGRAM

// ---- POUs/prgHouse.TcPOU
PROGRAM prgHouse
VAR
	fbKBusState					: FB_K_Bus_State;
	uint_KBusState				: UINT;							
	lrHousePower				: LREAL;								
	lrNetzEinspeisung			: LREAL;								
	lrBetriebMuellerBau			: LREAL;								
	fbGrid1						: FB_EM_Beckhoff_KL3403;  	//UV Müller Holzbau
	fbGrid2						: FB_EM_Beckhoff_KL3403;	//Abgang Direktmessung
	fbGrid3						: FB_EM_Beckhoff_KL3403;	//Produktion PV
	(*
	lrGrid_Voltage_L1  	AT %I* : LREAL;										
    lrGrid_Current_L1 	AT %I* : LREAL;	
	lrGrid_Power_L1		AT %I* : LREAL;		
	lrGrid_Voltage_L2  	AT %I* : LREAL;										
    lrGrid_Current_L2 	AT %I* : LREAL;	
	lrGrid_Power_L2		AT %I* : LREAL;
	lrGrid_Voltage_L3  	AT %I* : LREAL;										
    lrGrid_Current_L3 	AT %I* : LREAL;	
	lrGrid_Power_L3		AT %I* : LREAL;									
	ActivePowerTotal	AT %I* : LREAL;		
	Test					   : REAL;	
*)
	lrGrid_Voltage_L1  	AT %I* 	: REAL;										
    lrGrid_Current_L1 	AT %I* 	: REAL;	
	lrGrid_Power_L1		AT %I* 	: REAL;		
	lrGrid_Voltage_L2  	AT %I* 	: REAL;										
    lrGrid_Current_L2 	AT %I* 	: REAL;	
	lrGrid_Power_L2		AT %I* 	: REAL;
	lrGrid_Voltage_L3  	AT %I* 	: REAL;										
    lrGrid_Current_L3 	AT %I* 	: REAL;	
	lrGrid_Power_L3		AT %I* 	: REAL;									
	ActivePowerTotal	AT %I*	: REAL;							
								
END_VAR

//lrNetzEinspeisung := fbGrid1.stDataEMPower.lrPowerTotal + fbGrid2.stDataEMPower.lrPowerTotal - fbGrid3.stDataEMPower.lrPowerTotal;	

//lrBetriebMuellerBau := (ActivePowerTotal_1 + ActivePowerTotal_2 + ActivePowerTotal_3) - fbGrid1.stDataEMPower.lrPowerTotal;

//The mapping of this function must be linked with the K-Bus State in the E/A Part
fbKBusState(	uiKBusState_OUT=> , 
				b_Kbus_notOk=> , 
				word_ErrorCount=> );
				
				


(*
fbGrid1(
	bEnable:= FALSE, 
	bChannel1Invers:= FALSE, 
	bChannel2Invers:= FALSE, 
	bChannel3Invers:= FALSE, 
	uiCurrentTransformerRatioL1:= 400, 
	uiCurrentTransformerRatioL2:= 400, 
	uiCurrentTransformerRatioL3:= 400, 
	uiKBusState_IN:= fbKBusState.uiKBusState_OUT, 
	stDataEMPower=> , 
	stDataEMCounter=> , 
	stDataEMPowerRealTime=> , 
	stDataEMCounterRealTime=> , 
	diNrOfEM_OUT=> );
	
	
fbGrid2(
	bEnable:= FALSE, 
	bChannel1Invers:= FALSE, 
	bChannel2Invers:= FALSE, 
	bChannel3Invers:= FALSE, 
	uiCurrentTransformerRatioL1:= 400, 
	uiCurrentTransformerRatioL2:= 400, 
	uiCurrentTransformerRatioL3:= 400, 
	uiKBusState_IN:= , 
	stDataEMPower=> , 
	stDataEMCounter=> , 
	stDataEMPowerRealTime=> , 
	stDataEMCounterRealTime=> , 
	diNrOfEM_OUT=> );
	
fbGrid3(
	bEnable:= FALSE, 
	bChannel1Invers:= FALSE, 
	bChannel2Invers:= FALSE, 
	bChannel3Invers:= FALSE, 
	uiCurrentTransformerRatioL1:= 400, 
	uiCurrentTransformerRatioL2:= 400, 
	uiCurrentTransformerRatioL3:= 400, 
	uiKBusState_IN:= , 
	stDataEMPower=> , 
	stDataEMCounter=> , 
	stDataEMPowerRealTime=> , 
	stDataEMCounterRealTime=> , 
	diNrOfEM_OUT=> );
*)

END_PROGRAM
